FUNCTION_BLOCK FB_CoolingSystem_IO
VAR
	Inputs							AT %I*	:	ST_CoolingSystemInputs;
	Outputs							AT %Q* 	:	ST_CoolingSystemOutputs;
	ControlData: INT;
	ScalePressure: FB_CTRL_SCALE;
	PressureScaleParams: ST_CTRL_SCALE_PARAMS := (tTaskCycleTime := TIME#1ms, tCtrlCycleTime := TIME#1ms, fInMin := 0, fInMax := 4095, fOutMin := 0, fOutMax := 10);
	ScaleTemp: FB_CTRL_SCALE;
	TempScaleParams: ST_CTRL_SCALE_PARAMS;
	

	BattValveDelayTimer: TP := (PT := CoolingSystemParams.MaximumValveOperatingTime);
	FancoilValveDelayTimer: TP := (PT := CoolingSystemParams.MaximumValveOperatingTime);
	InvValveDelayTimer: TP := (PT := CoolingSystemParams.MaximumValveOperatingTime);
END_VAR

VAR_IN_OUT
	IO			:	ST_CoolingSystem_Control;
	Events		: 	ST_CoolingSystemEvents; 
END_VAR
VAR
	IdlePressureMeasurementDelay: ST_CoolingSystemEvents;
END_VAR



//Convert and scale pressure sensor data
{warning "TODO: FB_CTRLSCALE werkt nog niet"}
IO.r_CoolantPressure := (INT_TO_REAL(Inputs.CoolingLoopPressureSensor)/409.6);
//ScalePressure(fIn := Inputs.CoolingLoopPressureSensor, stParams:= PressureScaleParams, fOut=>IO.r_CoolantPressure);

IF (NOT IO.b_ACPumpEnable) AND (NOT IO.b_DCPumpEnable) THEN
	IO.r_CoolantIdlePressure := IO.r_CoolantPressure;
END_IF

//Cooling system pressure check. Lowest pressure will occur with pumps off.
//if this dips below the minimum pressure, the system has lost coolant and should be fixed.
Events.b_CoolingLoopIdlePressureWarning := (IO.r_CoolantPressure < CoolingSystemParams.MinimumSystemBasePressureWarningLevel);
Events.b_CoolingLoopIdlePressureError 	:= (IO.r_CoolantPressure < CoolingSystemParams.MinimumSystemBasePressureErrorLevel);

//Convert and scale coolant tank temperature data
{warning "TODO: FB_CTRLSCALE werkt nog niet"}
IO.r_CoolantTemperature := (INT_TO_REAL(Inputs.CoolingLoopTemperatureSensor)/40.96)-40;
//ScalePressure(fIn := Inputs.CoolingLoopTemperatureSensor, stParams:= TempScaleParams, fOut=>IO.r_CoolantTemperature);

//Pump control
Outputs.ACPumpEnable := IO.b_ACPumpEnable;
Outputs.DCPumpEnable := IO.b_DCPumpEnable;

//FanControl
Outputs.DCFanEnable := IO.b_DCFancoilEnable;


//Battloop valve control
//First set output and edge detectors. The edge detectors trigger a grace period in which the valve state is allowed to diverge from requested state
Outputs.BattLoopValveClose := IO.b_CloseBatteryLoopValve;

//Feedback is inverse from output. If they stay the same for too long --> Valve is stuck or inoperative
IO.b_BatteryLoopEnabled := Inputs.BattLoopValveFB;
BattValveDelayTimer(IN := IO.b_CloseBatteryLoopValve = Inputs.BattLoopValveFB);
Events.b_BattLoopValveStuck := BattValveDelayTimer.Q;


//Inverter loop valve control
//First set output and edge detectors. The edge detectors trigger a grace period in which the valve state is allowed to diverge from requested state
Outputs.InvLoopValveClose := IO.b_CloseInverterLoopValve;

//Feedback is inverse from output. If they stay the same for too long --> Valve is stuck or inoperative
IO.b_InverterLoopEnabled := Inputs.InvLoopValveFB;
InvValveDelayTimer(IN := IO.b_CloseInverterLoopValve = Inputs.InvLoopValveFB);
Events.b_InverterLoopValveStuck := InvValveDelayTimer.Q;


//Fancoil loop valve control
//First set output and edge detectors. The edge detectors trigger a grace period in which the valve state is allowed to diverge from requested state
Outputs.FancoilLoopValveClose := IO.b_CloseFancoilLoopValve;

//Feedback is inverse from output. If they stay the same for too long --> Valve is stuck or inoperative
IO.b_FancoilLoopEnabled := Inputs.FancoilLoopValveFB;
FancoilValveDelayTimer(IN := IO.b_CloseFancoilLoopValve = Inputs.FancoilLoopValveFB);
Events.b_FancoilLoopValveStuck := FancoilValveDelayTimer.Q;




//400V fuse feedback
Events.b_CoolingSystemFuseFailure := NOT Inputs.CoolingSystem400VFuseFB;

END_FUNCTION_BLOCK

(* stored: Version 1.1.0.1, ProductVersion 3.1.4024.12
   POU FB_CoolingSystem_IO: Id {ebb8c199-6485-481f-90e0-cc2169c528cd}, SpecialFunc None *)
